TYPE DriveStatus :
STRUCT
	ReadyToEnable : BOOL;
	Ready : BOOL;
	Warning : BOOL;
	Error : BOOL;
	MovingPositive : BOOL;
	MovingNegative : BOOL;
	DigitalInput1 : BOOL;
	DigitalInput2 : BOOL;
END_STRUCT
END_TYPE

(* stored: Version 1.1.0.1, ProductVersion 3.1.4024.9
   DUT DriveStatus: Id {68acc128-45ee-43eb-8ea7-016b493e8473} *)
